Xinje XDPPro project, PLC1: XDH-60T4 (software 3.7.14b 2022-06-24)

PROGRAM 梯形图

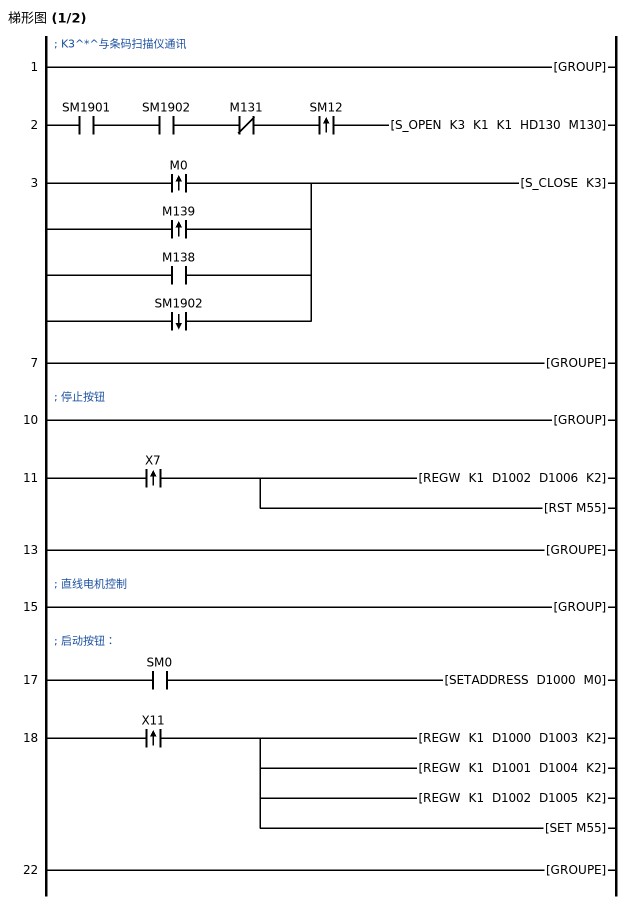
; K3^*^与条码扫描仪通讯
GROUP
LD     SM1901
AND    SM1902
ANI    M131
ANDP   SM12
S_OPEN K3 K1 K1 HD130 M130
LDP    M0
ORP    M139
OR     M138
ORF    SM1902
S_CLOSE K3
GROUPE
; 停止按钮
GROUP
LDP    X7
REGW   K1 D1002 D1006 K2
RST    M55
GROUPE
; 直线电机控制
GROUP
; 启动按钮：
LD     SM0
SETADDRESS D1000 M0
LDP    X11
REGW   K1 D1000 D1003 K2
REGW   K1 D1001 D1004 K2
REGW   K1 D1002 D1005 K2
SET    M55
GROUPE

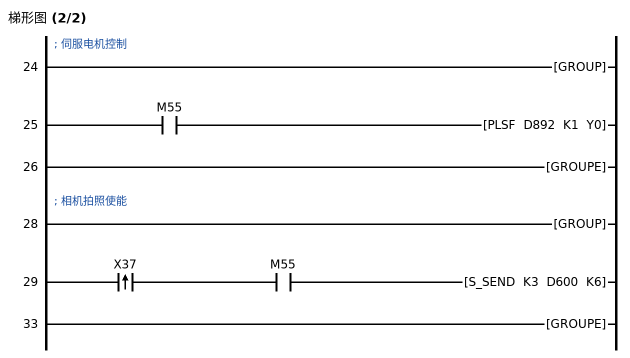
; 伺服电机控制
GROUP
LD     M55
PLSF   D892 K1 Y0
GROUPE
; 相机拍照使能
GROUP
LDP    X37
AND    M55
S_SEND K3 D600 K6
GROUPE

C FILE func1.h
#ifndef	_FUNC1_H
#define	_FUNC1_H
/*********宏定义用来存放需要的返回值************/
 //#define NEEDTIME D[3100]       //保存返回值
 //#define CAR      D[3102]        //存储判断出来的小车号
 //#define Bourn     D[3103]       //目的格口
 //#define Time      D[300]           //时间基点定时器的计数值 
#define D_D	     *(INT32S*)&D


/**********首地址************/
#define SendToLowPLCBuffAddress D+3100 //发送给分控的发送缓冲区首地址,总计15个寄存器
#define RCVDateFirstAddress D+2600      //上位机发来的数据缓冲区首地址，总计36个寄存器
#define SendACKToWCSFiestAddress D+3200 //向上位机回复ACK报文的数据缓冲区首地址，总计19个寄存器
#define SendToCameraFirstAddress D+600  //发给相机，6个寄存器
#define RCVDateFormLOW          D+2700  //分控分拣完成返回，24个寄存器
#define LOCKFIRSTADDRESS D+45000        //锁格队列首地址,101个寄存器
#define CarDateFirstAddress D+3300      //存放已有任务的小车数组


/* 存放一些函数中需要的参数 
所有的距离单位为毫米，时间单位为毫秒
 */
 
 
 #define TrackLength  50000         //轨道的长度
 #define  Speed  1                  //小车速度1mm/ms
 #define DistanceOfCar  400         //小车的间距(单位为：毫米)
 #define TIMELOSS  5                //电机启动时间偏移量(单位为：毫秒)

 #define Time_Offset 　0            //时间偏移量，由于没有进行实验测试暂时设置为0,该值是用来计算小车上的电机转动所需要的时间

 #define DistanceOfCut  750         //此处割口的间距 ————割口的长度加上割口间的距离

 #define  Camera_Position  600      //扫码设备->光电的距离
 #define Light2CameraPosition (TrackLength-Camera_Position)  //光电->扫码设备的距离

 #define Time  0                    //距离时间基点的时间

 
 #define SIZEOFLATTICE 100      //格口个数


//宏定义寄存器使用
#define PassedTime      D[888]
#define NowSpeed        D[890]         //皮带线当前速度
#define CarSpeed        D[891]         //小车线速度
#define PulseFrequency  D[892]   //皮带线脉冲频率
#define CarFrequency    D[893]   //小车线反馈脉冲频率
#define speedAddress     D[1000]  //Modbus转速地址
#define PowerAddress     D[1001]  //转矩地址
#define MasterAddress    D[1002]  //命令符地址
#define speedValue       D[1003]  //Modbus转速发送
#define PowerValue       D[1004]  //转矩发送
#define MasterValue      D[1005]  //命令符发送
#define StopMaster       D[1006]    //电机停止
#define CarIncConter   D[8801]  //小车线当前时间
#define PulseIncConter D[8800]  //皮带线当前计数值



#define CameraEnableTime D[894]     //相机使能定时时间
#define DZCL        D[8802]     //转一圈需要的脉冲数

#endif

C FUNCTION BLOCK setaddress.fcb
/* #EXPORT_ENTRY_BEGIN(SETADDRESS)
//    类型              模式             个数               映射          注释
W = { type = "PINT16S", mode = [In,Out], count = "unknown", map = [D,HD], comment = "" }
B = { type = "BIT"    , mode = [In,Out], count = "unknown", map = [M,HM], comment = "" }
#EXPORT_ENTRY_END */
/*************************************************************************
 * FunctionBlockName:  SETADDRESS
 * Version:            1.0.0
 * Author:             rpl
 * UpdateTime:         2022-08-25 16:03:02
 * Comment:            
**************************************************************************/

/**
 * @summary 
 * @param W 
 * @param B 
 */
#include"func1.h"
void SETADDRESS(PINT16S W,BIT B)
{
	#define SysRegAddr_HD_D_HM_M
    HM[10] = 1;
    speedAddress = 0x7002;
    PowerAddress = 0x7006;
    MasterAddress = 0x7000;
    speedValue  = 1000;
    PowerValue  = 1500;
    MasterValue = 1;
    StopMaster = 6;
    D[892] =speedValue/1.375*10;
    
    
    
    * ( SendToCameraFirstAddress ) = 0x02;
    //千位
    * ( SendToCameraFirstAddress + 1 ) = 0x30;
    //百位
    * ( SendToCameraFirstAddress + 2 ) = 48;
    //十位
    * ( SendToCameraFirstAddress + 3 ) = 48 ;
    //个位
    * ( SendToCameraFirstAddress + 4 ) = 48;
    //结束符
    * ( SendToCameraFirstAddress + 5 ) = 0x03;
    
    
    return;
}